{attribute 'GeneratedUsingTerminal: EL7031-0030-0016'}
{attribute addProperty BoxType "EL7031-0030-0016"}
{attribute addProperty Description "EL7031-0030 1Ch. Stepper motor output stage (24V, 2.8A)"}
{attribute addProperty Physics "KK"}
{attribute addProperty Id "ENC_Status_compactAT %I*ENC_Status_compact_3C6E2C4411STM_StatusAT %I*STM_Status_36ED096F11AI_Standard_Channel_1AT %I*AI_Standard_Channel_205D8A067AI_Standard_Channel_2AT %I*AI_Standard_Channel_205D8A067ENC_Control_compactAT %Q*ENC_Control_compact_2E82BC435STM_ControlAT %Q*STM_Control_5A8B50163STM_VelocityAT %Q*STM_Velocity_A47A3F412WcStateAT %I*WcState_9091E0EB2InfoDataAT %I*InfoData_939F71B614"}
{attribute addProperty CRC "3108784436"}
{attribute addProperty Size "62"}
TYPE EL7031_B94C4934 EXTENDS EtcSlaveTerminalBase_947E5A46 :
STRUCT
	{attribute addProperty Name "ENC_Status_compact"}
	ENC_Status_compact : ENC_Status_compact_3C6E2C44;
	{attribute addProperty Name "STM_Status"}
	STM_Status : STM_Status_36ED096F;
	{attribute addProperty Name "AI_Standard_Channel_1"}
	AI_Standard_Channel_1 : AI_Standard_Channel_205D8A06;
	{attribute addProperty Name "AI_Standard_Channel_2"}
	AI_Standard_Channel_2 : AI_Standard_Channel_205D8A06;
	{attribute addProperty Name "ENC_Control_compact"}
	ENC_Control_compact : ENC_Control_compact_2E82BC43;
	{attribute addProperty Name "STM_Control"}
	STM_Control : STM_Control_5A8B5016;
	{attribute addProperty Name "STM_Velocity"}
	STM_Velocity : STM_Velocity_A47A3F41;
	{attribute addProperty Name "WcState"}
	WcState : WcState_9091E0EB;
	{attribute addProperty Name "InfoData"}
	InfoData : InfoData_939F71B6;
END_STRUCT
END_TYPE

(* stored: Version 1.2.0.0, ProductVersion 3.1.4024.9
   DUT EL7031_B94C4934: Id {4763b7c0-9614-4076-a8f1-d4967d1d8fc3} *)
